(* PLC project v0.6.02_RefactorGateAndTest.project, CODESYS CODESYS V3.5 SP19 Patch 1 *)
(* stored: creationDateTime 2026-08-11T18:19:14.783359, modificationDateTime 2026-08-11T18:19:14.783359 *)

(* ═══════════════════════════════════════════════════════════════ 🧪 FB_Sim_Joystick — Simulation des entrées brutes joystick (bus CAN hors ligne) ─────────────────────────────────────────────────────────────── 📄 Doc métier : DOC/AF/AF_Partie-13_Fonction_Simulation_v2.1.md 🧩 Brique réduite (Partie3 §1bis) : outil de banc, pas du métier machine. 🎯 Rôle : remplace l'ancien bypass homme-mort codé en dur dans `FB_Joystick` (`GVL_DEBUG.DBG_DeadmanBypass_TEST`, qui forçait `DeadmanArmed` en permanence — un vrai contournement de sécurité). Ici, on simule les ENTRÉES BRUTES du capteur (`RawX`/`RawY`/`RawButton`) : le homme-mort réel de `FB_Joystick` reste pleinement actif et doit toujours être "actionné" (forcer `RawButton` en instance CODESYS) pour armer — comportement métier testé pour de vrai, pas contourné. 📥 Enable : simulation active (SimulationModeActive AND NOT BusJoystickSignalIsReal) — 🔧 REX 2026-07-08 : granularité séparée du bus CANopen (BusJoystickIsReal, voir GVL_Simulation) 📥 NeutralRaw : valeur brute simulée au repos (voir GVL_Simulation.TstJoystickForceNeutralRaw) 📥 MaxRaw : valeur brute simulée à fond (voir GVL_Simulation.TstJoystickForceMaxRaw) 📤 RawX/RawY : forçables en instance CODESYS (par défaut = NeutralRaw, repos) 📤 RawButton : forçable en instance CODESYS (par défaut = FALSE, relâché) 💡 Note d'application : en vue instance CODESYS, forcer `RawX`/`RawY` à `MaxRaw` (ou une valeur intermédiaire) pour simuler un débattement, et `RawButton` à `TRUE` pour simuler l'appui homme-mort — exactement comme on forcerait le vrai capteur. ═══════════════════════════════════════════════════════════════ === DECLARATION (à coller dans la partie déclaration du POU FB_Sim_Joystick) === *)
FUNCTION_BLOCK FB_Sim_Joystick
  VAR_INPUT
    Enable : BOOL;
    NeutralRaw : INT := 5000;
    MaxRaw : INT := 10000;
  END_VAR
  VAR_OUTPUT
    RawX : INT;  (* 🔧 Forçable en instance CODESYS (repos = NeutralRaw) *)
    RawY : INT;  (* 🔧 Forçable en instance CODESYS (repos = NeutralRaw) *)
    RawButton : BOOL;  (* 🔧 Forçable en instance CODESYS (repos = FALSE) *)
  END_VAR
  VAR
    FirstCycle : BOOL := TRUE;
  END_VAR

            

// === IMPLEMENTATION (à coller dans le corps ST du POU FB_Sim_Joystick) ===

// 🔑 Initialise au neutre au premier cycle uniquement — ensuite RawX/RawY/RawButton
// restent forçables librement en instance CODESYS (un Force n'est jamais écrasé par TRUE,
// mais une simple écriture cyclique l'écraserait — donc pas de ré-assignation continue ici).
IF NOT Enable THEN
    FirstCycle := TRUE;
    RETURN;
END_IF;

IF FirstCycle THEN
    RawX := NeutralRaw;
    RawY := NeutralRaw;
    RawButton := FALSE;
    FirstCycle := FALSE;
END_IF;

          
END_FUNCTION_BLOCK
